// Mitsubishi GX Works2 project: 240409_순시동작_복귀회로   PLC: Q03UDV

PROGRAM MAIN
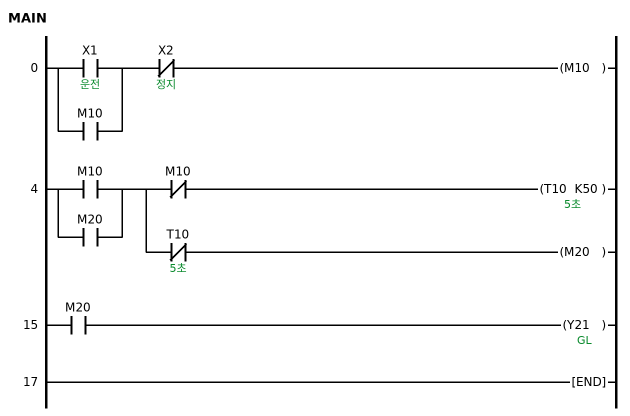
0     LD      X1  ; 운전
      OR      M10
      ANI     X2  ; 정지
      OUT     M10
4     LD      M10
      OR      M20
      MPS
      ANI     M10
      OUT     T10 K50  ; 5초
      MPP
      ANI     T10  ; 5초
      OUT     M20
15    LD      M20
      OUT     Y21  ; GL
17    END
END_PROGRAM

// device comments not shown above
X0  ; 정지
Y22  ; 정지
